TEXTLIST TextList_xyErrorid
  0 = 'no_error'
  1 = 'not_connected'
  2 = 'invalid_state'
  3 = 'actuator_out_of_pos_range'
  4 = 'actuator_out_of_neg_range'
  5 = 'homing_timeout'
  6 = 'parameter_out_of_range'
  7 = 'trigger_Limit'
  8 = 'SpeedNotReach'
  9 = 'homing_error'
  10 = 'cmd_timeout'
  11 = 'TBD_error'
  12 = 'io_error'
  13 = 'unknown_error'
  666 = 'emergency_error'
  14 = 'Drive_not_ready_for_operation'
  15 = 'interlock_error'
   = ''
END_TEXTLIST

(* stored: Version 1.1.0.1, ProductVersion 3.1.4024.11
   TextList TextList_xyErrorid: Id {246c0d90-1eba-4614-8703-4e5d5a47d843} *)
